{attribute 'linkalways'} 
{attribute 'no_explicit_call' := 'This FB is a CLASS and must be accessed using methods or properties'}
{attribute 'enable_dynamic_creation'}
FUNCTION_BLOCK Node_ContainerType_Vector_Vector_ULINT EXTENDS Node
VAR
    out : _GUID;
END_VAR

METHOD PUBLIC  Clone : I_Node
VAR
	pNode : POINTER TO Node_ContainerType_Vector_Vector_ULINT;
END_VAR
pNode := __NEW(Node_ContainerType_Vector_Vector_ULINT);
Clone := pNode^;
END_METHOD

METHOD FB_init : BOOL
VAR_INPUT
	bInitRetains : BOOL; // if TRUE, the retain variables are initialized (warm start / cold start)
	bInCopyCode : BOOL;  // if TRUE, the instance afterwards gets moved into the copy code (online change)
END_VAR
AddOutput('out', out);
END_METHOD

METHOD PROTECTED OnExecute
out.Value := ContainerType_Vector_Vector_ULINT;
END_METHOD

END_FUNCTION_BLOCK

(* stored: Version 1.1.0.1, ProductVersion 3.1.4026.17
   POU Node_ContainerType_Vector_Vector_ULINT: Id {718ca0bb-13e0-0d5e-1520-74e6c80a603f}, SpecialFunc None
   Folder Constructor: Id {c74032ea-1d9c-06b9-3e94-0cc6da79d350}
   Method Clone: Id {5404dbfe-c003-0a55-29aa-f1ca0f85e238}
   Method FB_init: Id {c8de75e7-b82f-0b24-3293-7293a8cd5a8d}
   Method OnExecute: Id {531dba73-0a57-0106-0e1c-04266ebe7623} *)
